Staubli VAL3: getSize.pgx

public program getSize(num& x_nSize[])
  local string l_sType
begin
  // give back the size to trajectory field
  x_nSize=size(pt:tTraj)
end
